// You will need Tc2_Math for this one
FUNCTION fnRoundLREAL_Method2 : LREAL
VAR_INPUT
	NumberToRound		:LREAL;		// Number that needs rounding
	Decimals			:USINT;		// Decimal places wanted
END_VAR
VAR
	rRoundREAL		:LREAL;
	rMultiplier		:LREAL;	
END_VAR

// Multiplier = 10^Decimals
rMultiplier := EXPT(10, Decimals);

// Shift decimal x positions to the right 
rRoundREAL := NumberToRound * rMultiplier;

// Round the number by converting it to an integer (use LINT for large numbers) 
rRoundREAL := LTRUNC(rRoundREAL);

// Shift decimal x potions back to the left
rRoundREAL := rRoundREAL / rMultiplier;

// Return result
fnRoundLREAL_Method2 := rRoundREAL;

END_FUNCTION

(* stored: Version 1.1.0.1, ProductVersion 3.1.4024.16
   POU fnRoundLREAL_Method2: Id {798d1f67-43a9-44cd-91d7-eaba9838cdcd}, SpecialFunc None *)
